// TwinCAT 3 PLC project PLC1
// Title: Bågsåg
// Company: JIAB
// Author: Johan Ivarsson
// ProjectVersion: 1.0.0
// Description: Testversion av en kap till MV teknik
// ProgramVersion: 3.1.4023.0
// libraries:
//   Tc2_MC2, * (Beckhoff Automation GmbH)
//   Tc2_MC2_Drive, * (Beckhoff Automation GmbH)
//   Tc2_Standard, * (Beckhoff Automation GmbH)
//   Tc2_System, * (Beckhoff Automation GmbH)
//   Tc2_Utilities, * (Beckhoff Automation GmbH)
//   Tc3_Module, * (Beckhoff Automation GmbH)
//   Tc3_EventLogger,3.1.30.0,Beckhoff Automation GmbH
//   VisuSymbols,3.5.10.0,System
// project tree:
//   10_Sekvens/ ST_Kapsekvens.TcPOU
//   20_Motion/ ST_Homing.TcPOU, ST_MotionControl.TcPOU
//   DUTs/ ST_MC_Status.TcDUT, ST_MC_CMD.TcDUT
//   / GlobalTextList.TcGTLO, PlcTask.TcTTO, Visualization Manager.TcVMO (not stored)
//   GVLs/ GVL.TcGVL, GVL_Motion.TcGVL
//   POUs/ LD_Spantransportor.TcPOU, MAIN.TcPOU
//   VISUs/ Visualization.TcVIS
// real-time tasks:
//   TASK PlcTask: cycle T#10ms, priority 20, ADS port 350
// motion (NC):
//   TASK NC-Task 1 SAF: cycle T#2ms, priority 4, ADS port 501
//   TASK NC-Task 1 SVB: cycle T#10ms, priority 8, ADS port 511
//   AXIS Y_Axis (id 1) // Matning till sågen
//     Velo: Maximum=2200
//     OtherSettings: AllowMotionCmdToSlave=true
//     encoder EncType=1
//     drive DrvType=5
//       Analog: TorqueSetpointScale=10, ScaleFactorActTorque=0.1
//       TimeComp: TaskDelayCycles=1
//     controller CtrType=1
//       CtrPara: PriorControlFactor=1
//         Observer: BandWidth=20
// variable links:
//   PLC1/PLC1 Instance <-> NC-Task 1 SAF/Axes/Y_Axis
//     PlcTask Inputs/GVL_Motion.Y_Axis.NcToPlc <-> Outputs/ToPlc
//     PlcTask Outputs/GVL_Motion.Y_Axis.PlcToNc <-> Inputs/FromPlc

CONFIGURATION PLC1
    RESOURCE PLC ON TwinCAT3
        TASK PlcTask(INTERVAL := T#10ms, PRIORITY := 20);
        PROGRAM MAIN WITH PlcTask : MAIN;
    END_RESOURCE
END_CONFIGURATION

// ---- DUTs/ST_MC_Status.TcDUT
TYPE ST_MC_Status :
STRUCT
	
	Status		: BOOL;
	Done		: BOOL;
	Busy		: BOOL;
	Error		: BOOL;
	Active		: BOOL;
	CmdAborted	: BOOL;
	InVelocity	: BOOL;
	ErrorID		: UDINt;
	
END_STRUCT
END_TYPE

// ---- DUTs/ST_MC_CMD.TcDUT
TYPE ST_MC_CMD :
STRUCT
	bExe				:	BOOL;
	lrVelocity			:	LREAL;
	lrAcceleration		:	LREAL;
	lrDeacceleration	:	LREAL;
	lrJerk				:	LREAL;
	lrDistance			:	LREAL;
	lrPosition			:	LREAL;
	enuDirection		:	MC_DIRECTION;
	enuBufferMode		:	MC_BUFFERMODE;
	enuOptions			:	ST_MOVEOPTIONS;
	
END_STRUCT
END_TYPE

// ---- GVLs/GVL.TcGVL
{attribute 'qualified_only'}
VAR_GLOBAL
	// Main funktioner //
	bPowerOn			:	BOOL;
	bPowerOff			:	BOOL;
	bEmergency			:	BOOL;
	bAutomaticMode		:	BOOL;
	bKapsekvens			:	BOOL;
	bKapsekvensDone		:	BOOL;

	// Svärd hållare //
	bSvard1				:	BOOL;
	bSvard2				:	BOOL;
	bSvardVentil1		:	BOOL;
	bSvardVentil2		:	BOOL;
	bSvard1Last			:	BOOL;
	bSvard1EjLast		:	BOOL;
	bSvard2Last			:	BOOL;
	bSvard2EjLast		:	BOOL;
	
	// Renhållning av maskin //
	bRenblasningsVentil	:	BOOL;
	Span_trans_Timer	: TOF;
	
	// Motor kontroller //
	bSagblad			:	BOOL;
	bKylpump			:	BOOL;
	
END_VAR

// ---- GVLs/GVL_Motion.TcGVL
{attribute 'qualified_only'}
VAR_GLOBAL
	// Singel axis GVL //
	
	Y_Axis	:	AXIS_REF;
	
	// Motion control funktionsblock //
	fbSA_Reset	:	MC_RESET;
	fbSA_Power	:	MC_POWER;
	fbSA_Home	:	MC_HOME;
	fbSA_Jog	:	MC_JOG;
	fbSA_MoveAbs1	:	MC_MoveAbsolute;
	fbSA_MoveAbs2	:	MC_MoveAbsolute;
	fbSA_SetPos		:	MC_SetPosition;
	
	fbSA_Halt		:	MC_HALT;
	fbSA_Stop		:	MC_STOP;
	
	// input: commands // 
	
	bSA_ResetExe		:	BOOL;
	bSA_HaltExe			:	BOOL;
	bSA_StopExe			:	BOOL;
	
	bSA_PowerEnCmd		:	BOOL;
	bSA_PowerEnPositive	:	BOOL:=TRUE;
	bSA_PowerEnNegative	:	BOOL:=TRUE;
	
	bSA_HomeExe			:	BOOL;
	bSA_HomeCamInput	:	BOOL;
	
	bSA_JogFwd			:	BOOL;
	bSA_JogRev			:	BOOL;
	
	stSA_AbsCmd1		:	ST_MC_CMD;
	stSA_AbsCmd2		:	ST_MC_CMD;
	
	// Variables/parameter //
	
	lrSA_PowerOverride	:	LREAL;
	lrSA_HomePosition	:	LREAL;
	lrSA_SetPosition	:	LREAL;
	lrSA_JogVelocity	:	LREAL;
	
	// Status //
	stSA_Reset	 		:	ST_MC_Status;
	stSA_Power		 	:	ST_MC_Status;
	stSA_Home		 	:	ST_MC_Status;
	stSA_SetPosition	:	ST_MC_Status;
	stSA_Jog			:	ST_MC_Status;
	
	stSA_AbsSts1		:	ST_MC_Status;
	stSA_AbsSts2		:	ST_MC_Status;
	
	stSA_Halt			:	ST_MC_Status;
	stSA_Stop			:	ST_MC_Status;
	

END_VAR

// ---- POUs/MAIN.TcPOU
PROGRAM MAIN
VAR
END_VAR

ST_MotionControl();
ST_Kapsekvens();
ST_Homing();
LD_Spantransportor();

END_PROGRAM

// ---- 20_Motion/ST_MotionControl.TcPOU
PROGRAM ST_MotionControl
VAR
END_VAR

LD_Y_AXIS_Sagning();

METHOD LD_Y_AXIS_Sagning : BOOL
VAR_INPUT
END_VAR

VAR
END_VAR
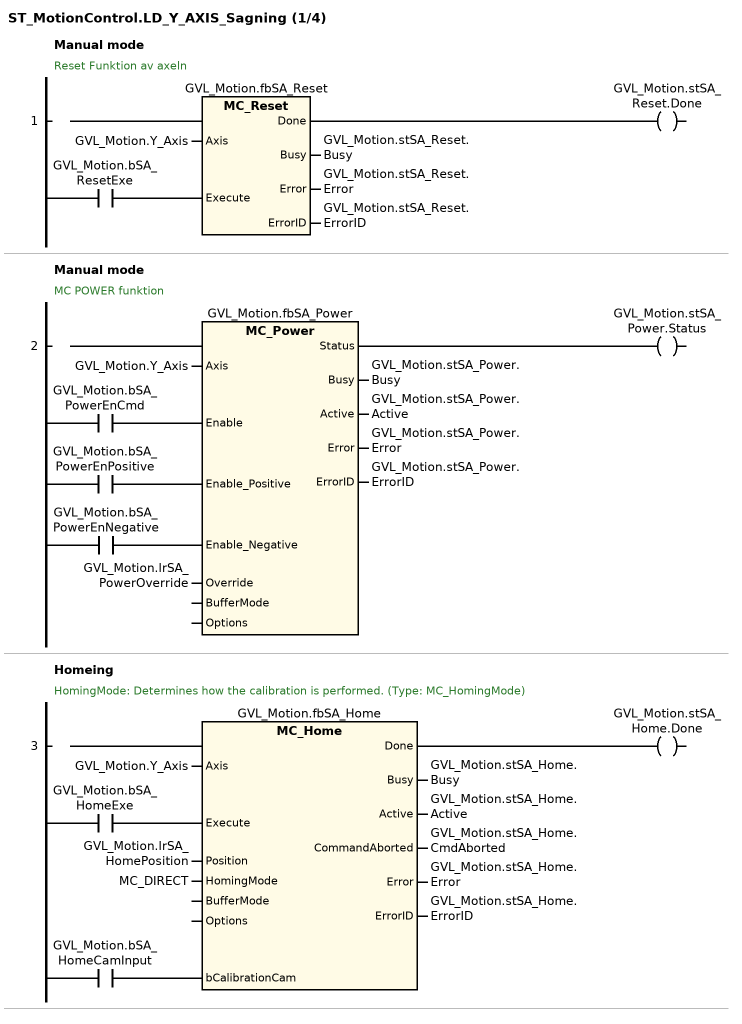
// NETWORK 1: Manual mode
// Reset Funktion av axeln
GVL_Motion.fbSA_Reset(
    Axis := GVL_Motion.Y_Axis,
    Execute := GVL_Motion.bSA_ResetExe,
    Busy => GVL_Motion.stSA_Reset.Busy,
    Error => GVL_Motion.stSA_Reset.Error,
    ErrorID => GVL_Motion.stSA_Reset.ErrorID); // MC_Reset
GVL_Motion.stSA_Reset.Done := GVL_Motion.fbSA_Reset.Done;

// NETWORK 2: Manual mode
// MC POWER funktion
GVL_Motion.fbSA_Power(
    Axis := GVL_Motion.Y_Axis,
    Enable := GVL_Motion.bSA_PowerEnCmd,
    Enable_Positive := GVL_Motion.bSA_PowerEnPositive,
    Enable_Negative := GVL_Motion.bSA_PowerEnNegative,
    Override := GVL_Motion.lrSA_PowerOverride,
    Busy => GVL_Motion.stSA_Power.Busy,
    Active => GVL_Motion.stSA_Power.Active,
    Error => GVL_Motion.stSA_Power.Error,
    ErrorID => GVL_Motion.stSA_Power.ErrorID); // MC_Power
GVL_Motion.stSA_Power.Status := GVL_Motion.fbSA_Power.Status;

// NETWORK 3: Homeing
// HomingMode: Determines how the calibration is performed. (Type: MC_HomingMode)
GVL_Motion.fbSA_Home(
    Axis := GVL_Motion.Y_Axis,
    Execute := GVL_Motion.bSA_HomeExe,
    Position := GVL_Motion.lrSA_HomePosition,
    HomingMode := MC_DIRECT,
    bCalibrationCam := GVL_Motion.bSA_HomeCamInput,
    Busy => GVL_Motion.stSA_Home.Busy,
    Active => GVL_Motion.stSA_Home.Active,
    CommandAborted => GVL_Motion.stSA_Home.CmdAborted,
    Error => GVL_Motion.stSA_Home.Error,
    ErrorID => GVL_Motion.stSA_Home.ErrorID); // MC_Home
GVL_Motion.stSA_Home.Done := GVL_Motion.fbSA_Home.Done;

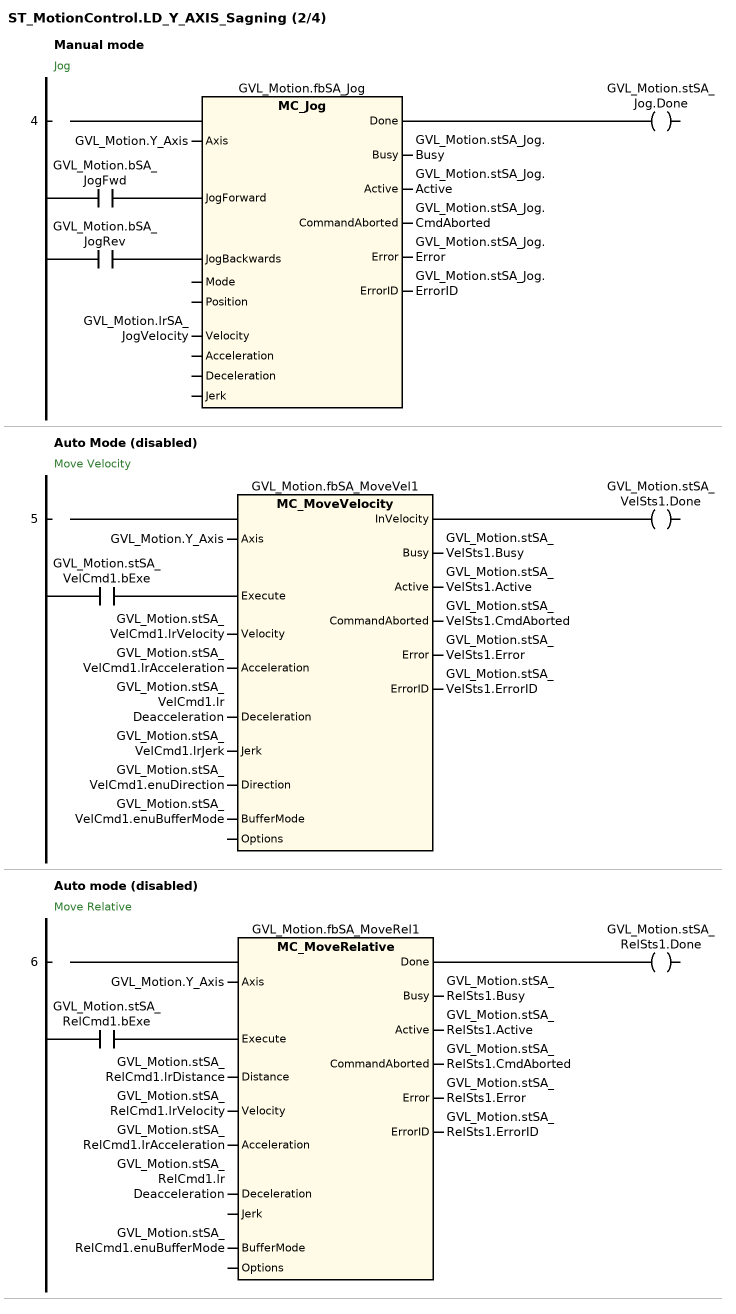
// NETWORK 4: Manual mode
// Jog
GVL_Motion.fbSA_Jog(
    Axis := GVL_Motion.Y_Axis,
    JogForward := GVL_Motion.bSA_JogFwd,
    JogBackwards := GVL_Motion.bSA_JogRev,
    Velocity := GVL_Motion.lrSA_JogVelocity,
    Busy => GVL_Motion.stSA_Jog.Busy,
    Active => GVL_Motion.stSA_Jog.Active,
    CommandAborted => GVL_Motion.stSA_Jog.CmdAborted,
    Error => GVL_Motion.stSA_Jog.Error,
    ErrorID => GVL_Motion.stSA_Jog.ErrorID); // MC_Jog
GVL_Motion.stSA_Jog.Done := GVL_Motion.fbSA_Jog.Done;

// NETWORK 5: Auto Mode (disabled)
// Move Velocity
// GVL_Motion.fbSA_MoveVel1(
//     Axis := GVL_Motion.Y_Axis,
//     Execute := GVL_Motion.stSA_VelCmd1.bExe,
//     Velocity := GVL_Motion.stSA_VelCmd1.lrVelocity,
//     Acceleration := GVL_Motion.stSA_VelCmd1.lrAcceleration,
//     Deceleration := GVL_Motion.stSA_VelCmd1.lrDeacceleration,
//     Jerk := GVL_Motion.stSA_VelCmd1.lrJerk,
//     Direction := GVL_Motion.stSA_VelCmd1.enuDirection,
//     BufferMode := GVL_Motion.stSA_VelCmd1.enuBufferMode,
//     Busy => GVL_Motion.stSA_VelSts1.Busy,
//     Active => GVL_Motion.stSA_VelSts1.Active,
//     CommandAborted => GVL_Motion.stSA_VelSts1.CmdAborted,
//     Error => GVL_Motion.stSA_VelSts1.Error,
//     ErrorID => GVL_Motion.stSA_VelSts1.ErrorID); // MC_MoveVelocity
// GVL_Motion.stSA_VelSts1.Done := GVL_Motion.fbSA_MoveVel1.InVelocity;

// NETWORK 6: Auto mode (disabled)
// Move Relative
// GVL_Motion.fbSA_MoveRel1(
//     Axis := GVL_Motion.Y_Axis,
//     Execute := GVL_Motion.stSA_RelCmd1.bExe,
//     Distance := GVL_Motion.stSA_RelCmd1.lrDistance,
//     Velocity := GVL_Motion.stSA_RelCmd1.lrVelocity,
//     Acceleration := GVL_Motion.stSA_RelCmd1.lrAcceleration,
//     Deceleration := GVL_Motion.stSA_RelCmd1.lrDeacceleration,
//     BufferMode := GVL_Motion.stSA_RelCmd1.enuBufferMode,
//     Busy => GVL_Motion.stSA_RelSts1.Busy,
//     Active => GVL_Motion.stSA_RelSts1.Active,
//     CommandAborted => GVL_Motion.stSA_RelSts1.CmdAborted,
//     Error => GVL_Motion.stSA_RelSts1.Error,
//     ErrorID => GVL_Motion.stSA_RelSts1.ErrorID); // MC_MoveRelative
// GVL_Motion.stSA_RelSts1.Done := GVL_Motion.fbSA_MoveRel1.Done;

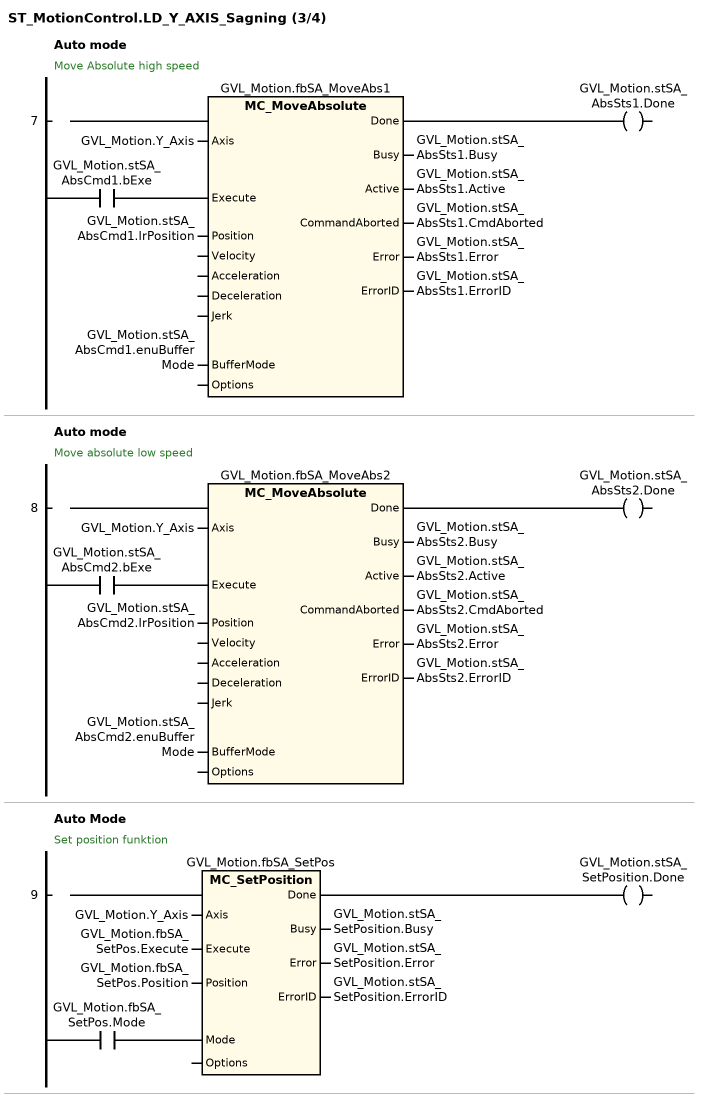
// NETWORK 7: Auto mode
// Move Absolute high speed
GVL_Motion.fbSA_MoveAbs1(
    Axis := GVL_Motion.Y_Axis,
    Execute := GVL_Motion.stSA_AbsCmd1.bExe,
    Position := GVL_Motion.stSA_AbsCmd1.lrPosition,
    BufferMode := GVL_Motion.stSA_AbsCmd1.enuBufferMode,
    Busy => GVL_Motion.stSA_AbsSts1.Busy,
    Active => GVL_Motion.stSA_AbsSts1.Active,
    CommandAborted => GVL_Motion.stSA_AbsSts1.CmdAborted,
    Error => GVL_Motion.stSA_AbsSts1.Error,
    ErrorID => GVL_Motion.stSA_AbsSts1.ErrorID); // MC_MoveAbsolute
GVL_Motion.stSA_AbsSts1.Done := GVL_Motion.fbSA_MoveAbs1.Done;

// NETWORK 8: Auto mode
// Move absolute low speed
GVL_Motion.fbSA_MoveAbs2(
    Axis := GVL_Motion.Y_Axis,
    Execute := GVL_Motion.stSA_AbsCmd2.bExe,
    Position := GVL_Motion.stSA_AbsCmd2.lrPosition,
    BufferMode := GVL_Motion.stSA_AbsCmd2.enuBufferMode,
    Busy => GVL_Motion.stSA_AbsSts2.Busy,
    Active => GVL_Motion.stSA_AbsSts2.Active,
    CommandAborted => GVL_Motion.stSA_AbsSts2.CmdAborted,
    Error => GVL_Motion.stSA_AbsSts2.Error,
    ErrorID => GVL_Motion.stSA_AbsSts2.ErrorID); // MC_MoveAbsolute
GVL_Motion.stSA_AbsSts2.Done := GVL_Motion.fbSA_MoveAbs2.Done;

// NETWORK 9: Auto Mode
// Set position funktion
GVL_Motion.fbSA_SetPos(
    Axis := GVL_Motion.Y_Axis,
    Execute := GVL_Motion.fbSA_SetPos.Execute,
    Position := GVL_Motion.fbSA_SetPos.Position,
    Mode := GVL_Motion.fbSA_SetPos.Mode,
    Busy => GVL_Motion.stSA_SetPosition.Busy,
    Error => GVL_Motion.stSA_SetPosition.Error,
    ErrorID => GVL_Motion.stSA_SetPosition.ErrorID); // MC_SetPosition
GVL_Motion.stSA_SetPosition.Done := GVL_Motion.fbSA_SetPos.Done;

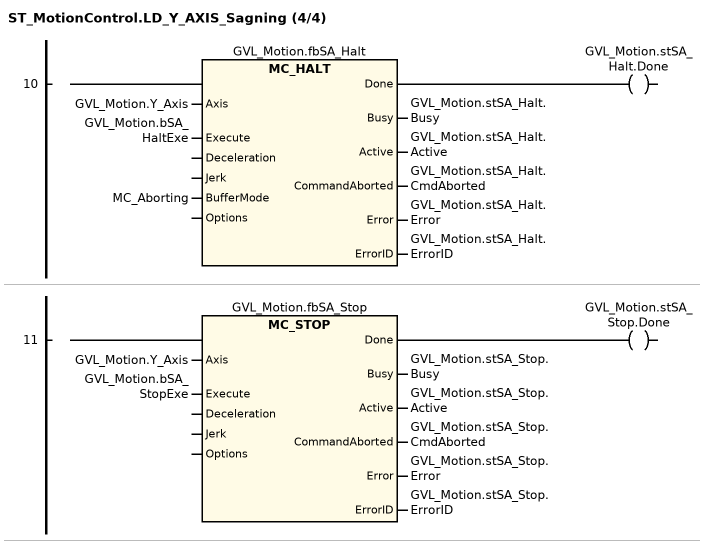
// NETWORK 10
GVL_Motion.fbSA_Halt(
    Axis := GVL_Motion.Y_Axis,
    Execute := GVL_Motion.bSA_HaltExe,
    BufferMode := MC_Aborting,
    Busy => GVL_Motion.stSA_Halt.Busy,
    Active => GVL_Motion.stSA_Halt.Active,
    CommandAborted => GVL_Motion.stSA_Halt.CmdAborted,
    Error => GVL_Motion.stSA_Halt.Error,
    ErrorID => GVL_Motion.stSA_Halt.ErrorID); // MC_HALT
GVL_Motion.stSA_Halt.Done := GVL_Motion.fbSA_Halt.Done;

// NETWORK 11
GVL_Motion.fbSA_Stop(
    Axis := GVL_Motion.Y_Axis,
    Execute := GVL_Motion.bSA_StopExe,
    Busy => GVL_Motion.stSA_Stop.Busy,
    Active => GVL_Motion.stSA_Stop.Active,
    CommandAborted => GVL_Motion.stSA_Stop.CmdAborted,
    Error => GVL_Motion.stSA_Stop.Error,
    ErrorID => GVL_Motion.stSA_Stop.ErrorID); // MC_STOP
GVL_Motion.stSA_Stop.Done := GVL_Motion.fbSA_Stop.Done;
END_METHOD

END_PROGRAM

// ---- 10_Sekvens/ST_Kapsekvens.TcPOU
PROGRAM ST_Kapsekvens
VAR
	Kapsekvens	:		INT		:=0;
	ErrorCode : WSTRING;
	ErrorNumber	:	UDINT;
END_VAR

// Påbörjan av kapsekvens //
IF GVL.bAutomaticMode AND GVL.bPowerOn AND NOT GVL.bPowerOff AND NOT GVL.bEmergency THEN
	Kapsekvens:=1;
ELSIF GVL.bEmergency OR GVL.bPowerOff THEN
	GVL_Motion.bSA_StopExe:=TRUE;
	GVL.bKylpump:=FALSE;
	GVL.bSagblad:=FALSE;
	GVL.bRenblasningsVentil:=FALSE;
	Kapsekvens:=2000;
END_IF

// Sekvens för sågning // 
CASE Kapsekvens	OF
	
	// Sekvens inom 1-9 är kontroll av program ect //
	1: IF GVL.bKapsekvens AND GVL.bAutomaticMode THEN
		Kapsekvens:=100;	
		ELSIF NOT GVL.bAutomaticMode THEN
			Kapsekvens:=2001;
		END_IF
		
	//Sekvens inom 100 inkulderar kontroll av svärd och låsning av det //
	100:IF GVL.bSvard1 THEN
			GVL.bSvard1Last:=TRUE; // För testning
			GVL.bSvard2Last:=TRUE; // För testning
			GVL.bSvard1EjLast:=FALSE; // För testning
			GVL.bSvard2EjLast:=FALSE; // För testning
			GVL.bSvardVentil1:=TRUE;
			GVL.bSvardVentil2:=TRUE;
			Kapsekvens:=110;
		ELSIF GVL.bSvard2 THEN
			GVL.bSvard1Last:=TRUE; // För testning
			GVL.bSvard2Last:=TRUE; // För testning
			GVL.bSvard1EjLast:=FALSE; // För testning
			GVL.bSvard2EjLast:=FALSE; // För testning
			GVL.bSvardVentil1:=TRUE;
			GVL.bSvardVentil2:=TRUE;
			Kapsekvens:=110;
		ELSE
			Kapsekvens:=2002;
		END_IF
	
	// Låsning av sågblad //	
	110: IF GVL.bSvard1Last THEN
			kapsekvens:=300;
		ELSIF GVL.bSvard2Last THEN
			kapsekvens:=300;
		ELSE
			Kapsekvens:=2003;
		END_IF
		
		
	(*// 200 är körning av sågblad/svärd till hemposition //
	//Påbörja homing //
	200: GVL_Motion.fbSA_Home(Axis:=GVL_Motion.Y_Axis,bCalibrationCam:=GVL_Motion.bSA_HomeCamInput,Execute:=TRUE);
		IF GVL_Motion.fbSA_Home.Busy THEN
			Kapsekvens:=210;
		END_IF
		
		
	// Homing pågår //
	210: IF GVL_Motion.fbSA_Home.Done AND NOT GVL_Motion.fbSA_Home.Error THEN
			GVL_Motion.bSA_HomeExe:=FALSE;
			Kapsekvens:=220;
		ELSIF GVL_Motion.stSA_Home.Error THEN
			GVL_Motion.bSA_HomeExe:=FALSE;
			Kapsekvens:=2003;
		END_IF
		
	// Homing klar //
	220: IF GVL_Motion.fbSA_Home.Done THEN
		Kapsekvens:=300;
		END_IF*)
		
	// Sekvens inom 300 är sågning av två blad //
	// Snabbkörning till kap pos //
	300:GVL.bSagblad:=TRUE;
		GVL.bKylpump:=TRUE;
		IF GVL.bSvard1Last AND GVL.bSvard2Last THEN
		 GVL_Motion.fbSA_MoveAbs1(Axis:=GVL_Motion.Y_Axis,
			Position := 100,
			Velocity := 50,
			Acceleration := 500,
			Deceleration := 500,
			Jerk := 100000,
			Execute:=TRUE);
			Kapsekvens:=310;
		ELSE
			Kapsekvens:=400;
		END_IF
	
		// pre-Positionerar kap //
	310:IF GVL_Motion.stSA_AbsSts1.Done AND NOT GVL_Motion.stSA_AbsSts1.Error THEN
			GVL_Motion.fbSA_MoveAbs1(Axis:=GVL_Motion.Y_Axis,Execute:=FALSE);
			Kapsekvens:=320;
		ELSIF GVL_Motion.stSA_AbsSts1.Error THEN
			GVL_Motion.fbSA_MoveAbs1(Axis:=GVL_Motion.Y_Axis,Execute:=FALSE);
			Kapsekvens:=2004;
		END_IF
		
		//Lågfarts matning när den arbetar i svärden //
	320: GVL_Motion.fbSA_MoveAbs2(Axis:=GVL_Motion.Y_Axis,
			Position := 200,
			Velocity := 5,
			Acceleration := 250,
			Deceleration := 250,
			Jerk := 100000,
			Execute:=TRUE);
		Kapsekvens:=330;
			
		// Kör till måldjup i svärden //
	330:IF GVL_Motion.stSA_AbsSts2.Done AND NOT GVL_Motion.stSA_AbsSts2.Error THEN
			GVL_Motion.fbSA_MoveAbs2(Axis:=GVL_Motion.Y_Axis,Execute:=FALSE);
			Kapsekvens:=500;
		ELSIF GVL_Motion.stSA_AbsSts2.Error THEN
			GVL_Motion.fbSA_MoveAbs2(Axis:=GVL_Motion.Y_Axis,Execute:=FALSE);
			Kapsekvens:=2005;
		END_IF
		
			
		
	// Sekvens inom 400 är sågning av ett blad //
	// Snabbkörning till kap pos //
	400:IF GVL.bSvard1Last OR GVL.bSvard2Last THEN
		 GVL_Motion.fbSA_MoveAbs1(Axis:=GVL_Motion.Y_Axis,
			Position := 100,
			Velocity := 50,
			Acceleration := 500,
			Deceleration := 500,
			Jerk := 100000,
			Execute:=TRUE);
		Kapsekvens:=410;
		ELSE
			Kapsekvens:=500;
		END_IF
	
		// pre-Positionerar kap //
	410:IF GVL_Motion.stSA_AbsSts1.Done AND NOT GVL_Motion.stSA_AbsSts1.Error THEN
			GVL_Motion.fbSA_MoveAbs1(Axis:=GVL_Motion.Y_Axis,Execute:=FALSE);
			Kapsekvens:=420;
		ELSIF GVL_Motion.stSA_AbsSts1.Error THEN
			GVL_Motion.fbSA_MoveAbs1(Axis:=GVL_Motion.Y_Axis,Execute:=FALSE);
			Kapsekvens:=2004;
		END_IF
		
		//Lågfarts matning när den arbetar i svärden //
	420: GVL_Motion.fbSA_MoveAbs2(Axis:=GVL_Motion.Y_Axis,
			Position := 200,
			Velocity := 10,
			Acceleration := 250,
			Deceleration := 250,
			Jerk := 100000,
			Execute:=TRUE);
		Kapsekvens:=430;
			
		// Kör till måldjup i svärden //
	430:IF GVL_Motion.stSA_AbsSts2.Done AND NOT GVL_Motion.stSA_AbsSts2.Error THEN
			GVL_Motion.fbSA_MoveAbs1(Axis:=GVL_Motion.Y_Axis,Execute:=FALSE);
			Kapsekvens:=500;
		ELSIF GVL_Motion.stSA_AbsSts2.Error THEN
			GVL_Motion.fbSA_MoveAbs2(Axis:=GVL_Motion.Y_Axis,Execute:=FALSE);
			Kapsekvens:=2005;
		END_IF
		
		
	// Sekvens inom 500 är Avslutad sågning //
	// Avslutad sågning //
	// Positionera såg //
	500: GVL_Motion.fbSA_MoveAbs1(Axis:=GVL_Motion.Y_Axis,
			Position := 0,
			Velocity := 400,
			Acceleration := 2500,
			Deceleration := 2500,
			Jerk := 100000,
			Execute:=TRUE);
		GVL.bRenblasningsVentil:=TRUE;
		GVL.bKapsekvensDone:=TRUE;
		Kapsekvens:=510;
	
	// Stäng av sågblad, kylning mm //
	510:GVL.bSagblad:=FALSE;
		GVL.bKylpump:=FALSE;
		GVL.bKapsekvensDone:=FALSE;
		GVL.bSvardVentil1:=FALSE;
		GVL.bSvardVentil2:=FALSE;
		GVL.bSvard1Last:=FALSE; // För testning
		GVL.bSvard2Last:=FALSE; // För testning
		GVL.bSvard1EjLast:=TRUE; // För testning
		GVL.bSvard2EjLast:=TRUE; // För testning
		IF GVL_Motion.stSA_AbsSts1.Done AND NOT GVL_Motion.stSA_AbsSts1.Error THEN
			GVL_Motion.fbSA_MoveAbs1(Axis:=GVL_Motion.Y_Axis,Execute:=FALSE);
			Kapsekvens:=1;
			GVL.bRenblasningsVentil:=FALSE;
		ELSIF GVL_Motion.stSA_AbsSts1.Error THEN
			GVL_Motion.fbSA_MoveAbs1(Axis:=GVL_Motion.Y_Axis,Execute:=FALSE);
			Kapsekvens:=2004;
			GVL.bRenblasningsVentil:=FALSE;
		END_IF
	
	// Stop servo //	
	900:GVL_Motion.fbSA_Stop(Axis:=GVL_Motion.Y_Axis,Execute:=TRUE);
		IF GVL_Motion.bSA_HomeCamInput THEN
			GVL_Motion.fbSA_Stop(Axis:=GVL_Motion.Y_Axis,Execute:=FALSE);
		END_IF
	
	// Sekvens över 2000 är error hantering //
	2000: ErrorCode:="Nödstop!"; 
	2001: ErrorCode:="Ej i automatik";
	2002: ErrorCode:="Maskin tom?";
	2003: ErrorCode:="Hem position ej nådd";
	2004: ErrorNumber:=GVL_Motion.stSA_AbsSts1.ErrorID;
	2005: ErrorNumber:=GVL_Motion.stSA_AbsSts2.ErrorID;
	
END_CASE

END_PROGRAM

// ---- 20_Motion/ST_Homing.TcPOU
PROGRAM ST_Homing
VAR
	Sekvens: INT;
END_VAR

CASE Sekvens OF
	//Påbörja homing //
	10: GVL_Motion.fbSA_Home(Axis:=GVL_Motion.Y_Axis,bCalibrationCam:=GVL_Motion.bSA_HomeCamInput,Execute:=TRUE);
		IF GVL_Motion.fbSA_Home.Busy THEN
			Sekvens:=210;
		END_IF
		
		
	// Homing pågår //
	20: IF GVL_Motion.fbSA_Home.Done AND NOT GVL_Motion.fbSA_Home.Error THEN
			GVL_Motion.bSA_HomeExe:=FALSE;
			Sekvens:=220;
		ELSIF GVL_Motion.stSA_Home.Error THEN
			GVL_Motion.bSA_HomeExe:=FALSE;
			Sekvens:=2003;
		END_IF
		
	// Homing klar //
	30: IF GVL_Motion.fbSA_Home.Done THEN
		Sekvens:=300;
		END_IF
END_CASE

END_PROGRAM

// ---- POUs/LD_Spantransportor.TcPOU
PROGRAM LD_Spantransportor
VAR
	Span_transportor: BOOL;
END_VAR

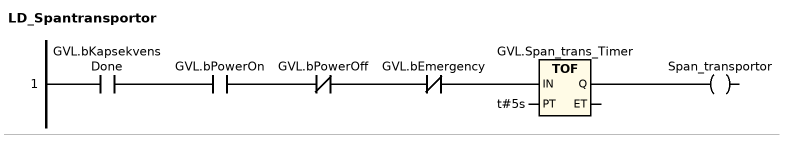
// NETWORK 1
GVL.Span_trans_Timer(IN := GVL.bKapsekvensDone AND GVL.bPowerOn AND NOT GVL.bPowerOff AND NOT GVL.bEmergency, PT := t#5s); // TOF
Span_transportor := GVL.Span_trans_Timer.Q;

END_PROGRAM

// ---- GlobalTextList.TcGTLO
TEXTLIST GlobalTextList
  785 = '%2.5f'
  475 = 'Akutell Position: %0.2f'
  868 = 'Akutell Position: %2.5f'
  540 = 'Akutell Position: %2f'
  814 = 'Automatic Mode'
  82 = 'CCCylinder'
  80 = 'ccyl ventil 2'
  462 = 'cyl ventil 1'
  558 = 'cyl ventil 2'
  115 = 'Cylinder'
  199 = 'Home position: %2.5f'
  819 = 'Home position: %f'
  58 = 'Homing'
  338 = 'Jog FWD'
  478 = 'Jog REV'
  717 = 'Kapsekvens: %0,3s'
  654 = 'Kapsekvens: %0.3s'
  904 = 'Kapsekvens: %3f'
  19 = 'Kylpump'
  579 = 'lås öpp'
  30 = 'Låst'
  837 = 'Nödstopp'
  477 = 'Override'
  420 = 'Power on'
  136 = 'Program start'
  290 = 'Renblås'
  312 = 'Reset'
  974 = 'Spån tr'
  629 = 'Spån trsp timer: %0.1s'
  176 = 'Spån trsp timer: %0.1s Sek'
  326 = 'Spån trsp timer: %1f'
  299 = 'Spån trsp timer: %1s'
  938 = 'Svärd 1'
  626 = 'Svärd 2'
  713 = 'Sågblad'
  467 = 'Öppen'
  421 = 'Öpppen'
END_TEXTLIST

// ---- VISUs/Visualization.TcVIS
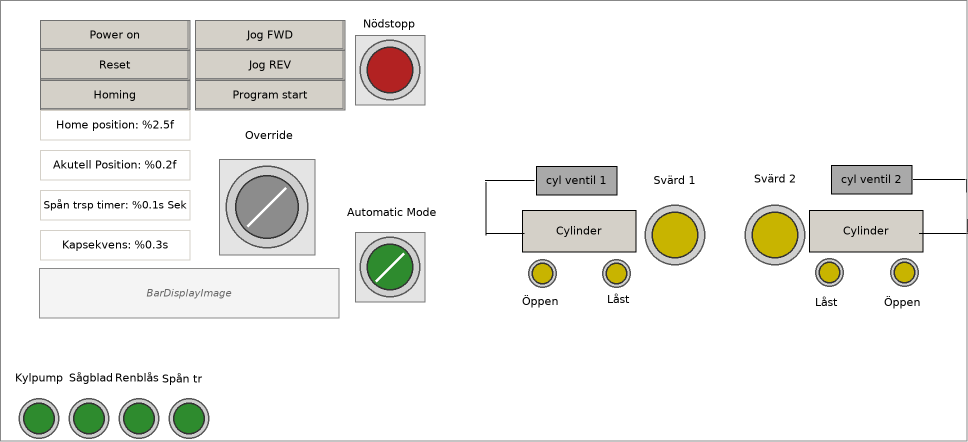
VISUALIZATION Visualization  // 968x442
    Potentiometer360 (219,157 96x100), variable: GVL_Motion.lrSA_PowerOverride, style: Potentiometer-Potentiometer360-Gray, scale format: %.1f, scale 0..100
        p2431819421: Outside
    BarDisplayImage (39,268 300x50), value: GVL_Motion.lrSA_PowerOverride, style: BarDisplayImage-Gray, scale format: %.1f, scale 0..100
    Button (40,20 150x30), "Power on"
        toggle GVL_Motion.bSA_PowerEnCmd
    Button (195,20 150x30), "Jog FWD"
        tap GVL_Motion.bSA_JogFwd
    Button (195,50 150x30), "Jog REV"
        tap GVL_Motion.bSA_JogRev
    Textfield (40,150 150x30), "Akutell Position: %0.2f", text variable: GVL_Motion.Y_Axis.NcToPlc.ActPos
    Button (40,50 150x30), "Reset"
        tap GVL_Motion.bSA_ResetExe
    Button (40,80 150x30), "Homing"
        tap GVL_Motion.bSA_HomeExe
    Textfield (40,110 150x30), "Home position: %2.5f", text variable: GVL_Motion.lrSA_HomePosition
    RotarySwitch (355,232 70x70), variable: GVL.bAutomaticMode, behaviour: TOGGLE, style: Switch-RotarySwitch-Green
    Button (195,80 150x30), "Program start"
        tap GVL.bKapsekvens
    Label (198,117 142x37), "Override"
    Textfield (40,190 150x30), "Spån trsp timer: %0.1s Sek", text variable: GVL.Span_trans_Timer.ET
    Textfield (40,230 150x30), "Kapsekvens: %0.3s", text variable: ST_Kapsekvens.Kapsekvens
    Lamp1 (15,395 48x47), variable: GVL.bKylpump, style: Lamp-Lamp1-Green
    Lamp1 (65,395 48x47), variable: GVL.bSagblad, style: Lamp-Lamp1-Green
    Label (56,363 70x30), "Sågblad"
    Label (4,363 70x30), "Kylpump"
    Label (321,194 142x37), "Automatic Mode"
    Lamp1 (115,395 48x47), variable: GVL.bRenblasningsVentil, style: Lamp-Lamp1-Green
    Label (102,363 70x30), "Renblås"
    Lamp1 (640,200 70x70), variable: GVL.bSvard1, style: Lamp-Lamp1-Yellow
    Lamp1 (740,200 70x70), variable: GVL.bSvard2, style: Lamp-Lamp1-Yellow
    Label (642,165 65x31), "Svärd 1"
    Label (742,160 66x38), "Svärd 2"
    Lamp1 (813,256 33x33), variable: GVL.bSvard2Last, style: Lamp-Lamp1-Yellow
    Lamp1 (888,256 33x33), variable: GVL.bSvard2EjLast, style: Lamp-Lamp1-Yellow
    Lamp1 (526,257 33x33), variable: GVL.bSvard1EjLast, style: Lamp-Lamp1-Yellow
    Lamp1 (600,257 33x33), variable: GVL.bSvard1Last, style: Lamp-Lamp1-Yellow
    Rectangle (522,210 114x42), "Cylinder"
    Rectangle (809,210 114x42), "Cylinder"
    Rectangle (831,165 81x29), "cyl ventil 2"
        p2257300284: GVL.bSvardVentil2
    Rectangle (536,166 81x29), "cyl ventil 1"
        p2257300284: GVL.bSvardVentil1
    Line (915,175)
    Line (913,179) (965,179)
    Line (966,179) (967,232)
    Line (919,233) (968,233)
    Line (485,180) (534,180)
    Line (486,233) (524,233)
    Line (486,235) (486,182)
    Label (508,286 65x31), "Öppen"
    Label (586,284 65x31), "Låst"
    Label (794,287 65x31), "Låst"
    Label (870,287 65x31), "Öppen"
    Lamp1 (165,395 48x47), variable: LD_Spantransportor.Span_transportor, style: Lamp-Lamp1-Green
    Label (147,364 70x30), "Spån tr"
    PushSwitch (355,35 70x70), variable: GVL.bEmergency, behaviour: TOGGLE, style: Switch-PushSwitch-Red
    Label (342,10 94x28), "Nödstopp"
END_VISUALIZATION
